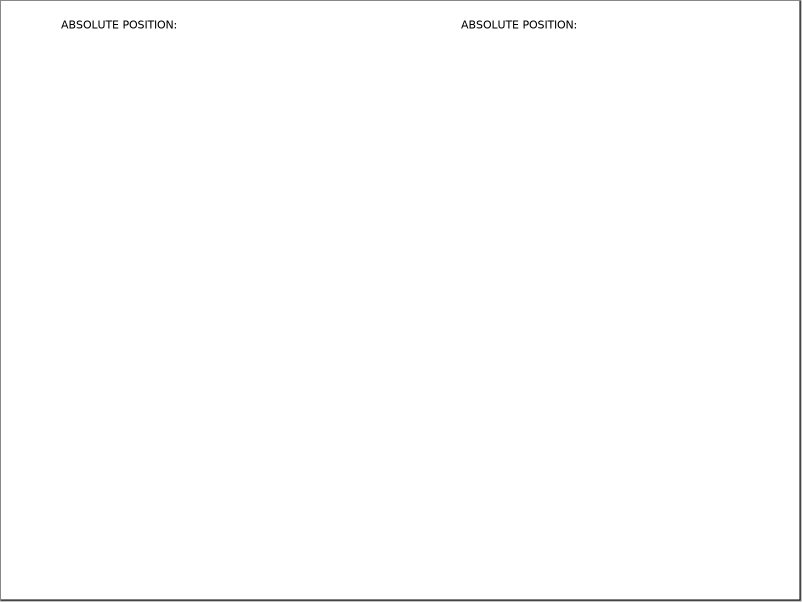
VISUALIZATION F47_Cam_In  // 802x602
    Rectangle (0,0 800x600)
    Label (10,10 170x30), "ABSOLUTE POSITION:"
    Label (410,10 170x30), "ABSOLUTE POSITION:"
END_VISUALIZATION

(* stored: Version 1.1.0.1, ProductVersion 3.1.4022.7
   Visu F47_Cam_In: Id {0484b24b-f68f-45a8-9eed-25b0bb9c396e} *)
